# B&R Automation Studio project Project
Automation Studio 4.9

## Configuration Config1

CPU X20CP3586, AutomationRuntime J4.93, Build 4.1.2, Safety 0.0, Vc V4.73.2

### Hardware
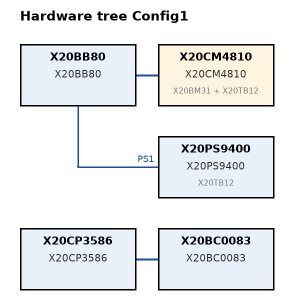
```
X20BB80 : X20BB80 v1.1.0.0
X20BC0083 : X20BC0083 v2.14.0.0  [PLK1 -> X20CP3586.IF3 (NodeNumber=1) [Cable Type=PowerlinkCable, Length=10, Version=1.0.0.3]; SL -> X20BB80.SL1]
  EnableDNA = on
X20BM31 : X20BM31 v1.1.0.0  [X2X1 -> X20BB80.IF1]
X20CM4810 : X20CM4810 v1.7.0.0  [SS1 -> X20TB12a.SS; SL -> X20BM31.SL1]
  Current01 = on
  CalcVel01 = on
  FLOWQ01 = 16#0002
  AICalc01 = on
  AIParameter01 = PEAK
  Current02 = on
X20CP3586 : X20CP3586 v1.10.0.0
  Connector IF2:
    ActivateDevice = 1
    HostName = cotrace-api
    Mode = Manual
    InternetAddress = 10.24.137.37
    SubnetMask = 255.255.255.0
  Connector IF3:
    EplHostName = cotrace-api
    HostName = cotrace-api
  ConfigurationID = CoTrace_Vibor_Config1
  VolatileGlobalPvSize = 200000
  IdleTaskClass = 1
  Cyclic1Duration = 2000
  Cyclic1Tolerance = 2000
  Cyclic3Duration = 48000
  Cyclic3Tolerance = 48000
  Cyclic8Duration = 8000
  Cyclic8Tolerance = 50000000
  Cyclic8Stack = 65000
  FileDevice1
  FileDeviceName1 = BufferData
  FileDevicePath1 = F:/BufferData
  EthernetHostName = cotrace-api
  EthernetDefaultGateway = 10.24.137.1
  FTPProtocol = 3
  FtpUser1
  FtpUsername1 = user
  FtpUserPassword1 = ztK7XSEqskzSOCpiuLWoesyAqwvBD/N0feCBZVSbf+w=
  FtpUserSalt1 = 7xprmDrz
  FTPAccessRight1 = 0
  WebServerProtocol = 2
  ActivateOpcUa = 1
  OpcUaInformationModels_PV_Version = 1
X20PS9400 : X20PS9400 v1.8.0.0  [SS1 -> X20TB12.SS; PS -> X20BB80.PS1]
X20TB12 : X20TB12 v1.0.0.0
X20TB12a : X20TB12 v1.0.0.0
```

### Hardware.hw.as4
```
Module X20BB80 (Type=X20BB80, Version=1.1.0.0)
Module X20BC0083 (Type=X20BC0083, Version=2.15.0.0)
  Connection (Connector=PLK1, TargetModule=X20CP3586, TargetConnector=IF3, NodeNumber=1)
    Cable (Type=PowerlinkCable, Length=10, Version=1.0.0.3)
  Connection (Connector=SL, TargetModule=X20BB80, TargetConnector=SL1)
Module X20BM31 (Type=X20BM31, Version=1.1.0.0)
  Connection (Connector=X2X1, TargetModule=X20BB80, TargetConnector=IF1)
Module X20CM4810 (Type=X20CM4810, Version=1.7.0.0)
  Connection (Connector=SS1, TargetModule=X20TB12a, TargetConnector=SS)
  Connection (Connector=SL, TargetModule=X20BM31, TargetConnector=SL1)
  Current01 = on
  CalcVel01 = on
  FLOWQ01 = 16#0002
  AICalc01 = on
  AIParameter01 = PEAK
  Current02 = on
Module X20CP3586 (Type=X20CP3586, Version=1.10.0.0)
  Connector IF2:
    ActivateDevice = 1
    HostName = cotrace-api
    Mode = Manual
    InternetAddress = 10.24.137.37
    SubnetMask = 255.255.255.0
  Connector IF3:
    EplHostName = cotrace-api
    HostName = cotrace-api
  ConfigurationID = CoTrace_Vibor_Config1
  Cyclic8Stack = 64000
  FileDevice1
  FileDeviceName1 = CoTraceWebApiFolder
  FileDevicePath1 = F:/CoTraceWebApiFolder
  FileDevice2
  FileDeviceName2 = SvgData
  FileDevicePath2 = F:/SvgData
  EthernetHostName = cotrace-api
  EthernetDefaultGateway = 10.24.137.1
  FTPProtocol = 3
  FtpUser1
  FtpUsername1 = user
  FtpUserPassword1 = ztK7XSEqskzSOCpiuLWoesyAqwvBD/N0feCBZVSbf+w=
  FtpUserSalt1 = 7xprmDrz
  FTPAccessRight1 = 0
  WebServerProtocol = 2
  ActivateOpcUa = 1
  OpcUaInformationModels_PV_Version = 1
Module X20PS9400 (Type=X20PS9400, Version=1.8.0.0)
  Connection (Connector=SS1, TargetModule=X20TB12, TargetConnector=SS)
  Connection (Connector=PS, TargetModule=X20BB80, TargetConnector=PS1)
Module X20TB12 (Type=X20TB12, Version=1.0.0.0)
Module X20TB12a (Type=X20TB12, Version=1.0.0.0)
```

### IoMap.iom - X20CP3586/IoMap.iom
```iecst
VAR_CONFIG
	::GetBuffer:fubCM4810.ioMapping.BufferInputSequence01 AT %IB."X20CM4810".BufferInputSequence01;
	::GetBuffer:fubCM4810.ioMapping.BufferRxByte01 AT %IB."X20CM4810".BufferRxByte01;
	::GetBuffer:fubCM4810.ioMapping.BufferRxByte02 AT %IB."X20CM4810".BufferRxByte02;
	::GetBuffer:fubCM4810.ioMapping.BufferRxByte03 AT %IB."X20CM4810".BufferRxByte03;
	::GetBuffer:fubCM4810.ioMapping.BufferRxByte04 AT %IB."X20CM4810".BufferRxByte04;
	::GetBuffer:fubCM4810.ioMapping.BufferRxByte05 AT %IB."X20CM4810".BufferRxByte05;
	::GetBuffer:fubCM4810.ioMapping.BufferOutputSequence01 AT %QB."X20CM4810".BufferOutputSequence01;
	::GetBuffer:fubCM4810.ioMapping.BufferTxByte01 AT %QB."X20CM4810".BufferTxByte01;
	::GetBuffer:fubCM4810.ioMapping.BufferTxByte02 AT %QB."X20CM4810".BufferTxByte02;
	::GetBuffer:fubCM4810.ioMapping.BufferTxByte03 AT %QB."X20CM4810".BufferTxByte03;
	::GetBuffer:fubCM4810.ioMapping.BufferTxByte04 AT %QB."X20CM4810".BufferTxByte04;
	::GetBuffer:fubCM4810.ioMapping.BufferLockValid01 AT %IX."X20CM4810".BufferLockValid01;
	::GetBuffer:fubCM4810.ioMapping.RequestBufferLock01 AT %QX."X20CM4810".RequestBufferLock01; (* SensorData[1] - CM4810 Channel 1 *)
	::SensorData[1].RmsAccRaw AT %ID."X20CM4810".RmsAccRaw01;
	::SensorData[1].RmsAccEnvelope AT %ID."X20CM4810".RmsAccEnvelope01;
	::SensorData[1].RmsVelRaw AT %ID."X20CM4810".RmsVelRaw01;
	::SensorData[1].RmsVelEnvelope AT %ID."X20CM4810".RmsVelEnvelope01;
	::SensorData[1].KurtosisRaw AT %ID."X20CM4810".KurtosisRaw01;
	::SensorData[1].SkewnessRaw AT %ID."X20CM4810".SkewnessRaw01;
	::SensorData[1].Vdi3832KtRaw AT %ID."X20CM4810".Vdi3832KtRaw01;
	::SensorData[1].ActSpeed AT %ID."X20CM4810".ActSpeed01;
	::SensorData[2].RmsAccRaw AT %ID."X20CM4810".RmsAccRaw02;
	::SensorData[2].RmsAccEnvelope AT %ID."X20CM4810".RmsAccEnvelope02;
	::SensorData[2].RmsVelRaw AT %ID."X20CM4810".RmsVelRaw02;
	::SensorData[2].RmsVelEnvelope AT %ID."X20CM4810".RmsVelEnvelope02;
	::SensorData[2].KurtosisRaw AT %ID."X20CM4810".KurtosisRaw02;
	::SensorData[2].SkewnessRaw AT %ID."X20CM4810".SkewnessRaw02;
	::SensorData[2].Vdi3832KtRaw AT %ID."X20CM4810".Vdi3832KtRaw02;
	::SensorData[2].ActSpeed AT %ID."X20CM4810".ActSpeed02;
	::SensorData[3].RmsAccRaw AT %ID."X20CM4810".RmsAccRaw03; (*RMS Value of the acceleration raw signal from MinFrequencyRaw to MaxFrequencyRaw [mg], channel 2*)
	::SensorData[3].RmsVelEnvelope AT %ID."X20CM4810".RmsVelEnvelope03; (*RMS Value of the velocity envelope signal from MinFrequencyEnvelope to MaxFrequencyEnvelope [mm/s], channel 3 (0 = calculation of velocity signal is disabled)*)
	::SensorData[3].KurtosisRaw AT %ID."X20CM4810".KurtosisRaw03; (*Kurtosis (4th statistical moment) of the raw signal from 0 Hz to MaxFrequencyRaw [1], channel 3*)
	::SensorData[3].Vdi3832KtRaw AT %ID."X20CM4810".Vdi3832KtRaw03; (*Ratio of the refernce values to the actual measured values of the raw signal as defined in VDI 3832 [1], channel 3*)
	::SensorData[3].SkewnessRaw AT %ID."X20CM4810".SkewnessRaw03; (*Skewnes (3rd statistical moment) of the raw signal from 0 Hz to MaxFrequencyRaw [1], channel 3*)
	::SensorData[3].RmsAccEnvelope AT %ID."X20CM4810".RmsAccEnvelope03; (*RMS Value of the acceleration envelope signal from MinFrequencyEnvelope to MaxFrequencyEnvelope [mg], channel 2*)
	::SensorData[3].RmsVelRaw AT %ID."X20CM4810".RmsVelRaw03; (*RMS Value of the velocity raw signal from MinFrequencyRaw to MaxFrequencyRaw [mm/s], channel 2 (0 = calculation of velocity signal is disabled)*)
	::SensorData[4].RmsAccRaw AT %ID."X20CM4810".RmsAccRaw04;
	::SensorData[4].RmsAccEnvelope AT %ID."X20CM4810".RmsAccEnvelope04;
	::SensorData[4].RmsVelRaw AT %ID."X20CM4810".RmsVelRaw04;
	::SensorData[4].RmsVelEnvelope AT %ID."X20CM4810".RmsVelEnvelope04;
	::SensorData[4].KurtosisRaw AT %ID."X20CM4810".KurtosisRaw04;
	::SensorData[4].SkewnessRaw AT %ID."X20CM4810".SkewnessRaw04;
	::SensorData[4].Vdi3832KtRaw AT %ID."X20CM4810".Vdi3832KtRaw04;
	::SensorData[1].ActSpeed AT %QD."X20CM4810".ActSpeed01;
	::SensorData[2].ActSpeed AT %QD."X20CM4810".ActSpeed02;
	::SensorData[3].ActSpeed AT %QD."X20CM4810".ActSpeed03;
	::SensorData[4].ActSpeed AT %QD."X20CM4810".ActSpeed04;
END_VAR
```

## Logical view

Binary libraries used (declarations not repeated): FileIO, runtime, sys_lib, AsBrStr, AsIOVib, AsFltGen, brsystem, AsIOAcc

### Global.typ - Global data types
```iecst
(* ============================================================ *)
(* CM4810 SENSOR CHANNEL DATA - Mapped from X20CM4810 process data via IoMap *)

TYPE
	SensorChannelData : 	STRUCT
		RmsAccRaw : REAL;			(* RMS acceleration raw [g] *)
		RmsAccEnvelope : REAL;		(* RMS acceleration envelope [g] *)
		RmsVelRaw : REAL;			(* RMS velocity raw [mm/s] *)
		RmsVelEnvelope : REAL;		(* RMS velocity envelope [mm/s] *)
		KurtosisRaw : REAL;			(* Kurtosis raw [-] *)
		SkewnessRaw : REAL;			(* Skewness raw [-] *)
		Vdi3832KtRaw : REAL;		(* VDI3832 Kt raw [-] *)
		ActSpeed : REAL;			(* Actual speed [rpm] *)
	END_STRUCT;
END_TYPE

(* ============================================================ *)
(* CSV EXPORT STATE MACHINE - Single state variable for GetBuffer <-> SaveData communication*)

TYPE
	CSVExportState :
		(
		CSV_IDLE := 0, (* Waiting for export request *)
		CSV_REQUESTED := 1, (* GetBuffer requested export *)
		CSV_PROCESSING := 2, (* SaveData is exporting *)
		CSV_COMPLETED := 3, (* Export done, CSV ready *)
		CSV_ERROR := 4 (* Export failed *)
		);
END_TYPE

(* ============================================================ *)
(* OPC UA COMMAND INTERFACE [API -> PLC] - Write these variables from FastAPI to configure the job*)

TYPE
	BufferUploadCmd : 	STRUCT
		WorkID : STRING[80] := 'debug_123'; (* Unique job ID: "mach5_sens12_1234567890_raw" *)
		ModulePath : STRING[30] := 'IF3.ST1.IF1.ST2'; (* "IF3.ST1.IF1.ST2" - X2X module path *)
		BufferNumber : USINT := 66; (* Buffer to download: 9,11,13,15,25,27,29,31,66,67,70,71... *)
		BufferLength : UDINT := 4097; (* Number of values: 4097, 8193, or 65535 *)
		Start : BOOL := 0; (* Edge trigger - set TRUE to start job *)
		Reset : BOOL := 0; (* Edge trigger - set TRUE to reset after Done *)
	END_STRUCT;
END_TYPE

(* ============================================================ *)
(* OPC UA STATUS INTERFACE [PLC -> API] - Read these variables from FastAPI to monitor job progress*)

TYPE
	BufferUploadStatus : 	STRUCT
		CurrentWorkID : STRING[80]; (* Currently processing WorkID *)
		Busy : BOOL := 0; (* TRUE when PLC is working on a job *)
		Done : BOOL := 0; (* TRUE when job completed (CSV ready on FTP) *)
		Error : BOOL := 0; (* TRUE if error occurred *)
		ErrorID : UINT := 0; (* Error code from vbioCM4810.status or custom error *)
		Progress : USINT := 0; (* Job progress: 0-100% *)
		CSVFileName : STRING[100]; (* Name of generated CSV file *)
	END_STRUCT;
END_TYPE

(* ============================================================ *)
(* MAIN STRUCTURE - Global variable gTrace*)

TYPE
	TraceVibro : 	STRUCT  (* OPC UA Interface - API <-> PLC *)
		BufferUpload : BufferUploadCmd;
		BufferStatus : BufferUploadStatus; (* Internal communication - GetBuffer <-> SaveData *)
		CSVExport : CSVExportState; (* Single state variable: IDLE/REQUESTED/PROCESSING/COMPLETED/ERROR *) (* Buffer data storage - max 8193 values *) (* Note: Most CM4810 buffers use 8193 values. Only special cases use 65535. *)
		xAxis : ARRAY[0..8192]OF REAL;
		yAxis : ARRAY[0..8192]OF REAL;
	END_STRUCT;
END_TYPE
```

### Global.var - Global variables
```iecst
VAR
	gTrace : TraceVibro;
	SensorData : ARRAY[1..4] OF SensorChannelData;
END_VAR
```


### Program Logical/VibroBuffer/GetBuffer (IEC)

#### Variables.var
```iecst
VAR
	fubCM4810 : vbioCM4810; (* Function block for accessing the buffers of a CM4810 module *)
	bInitialized : BOOL := FALSE;
	stMachine : UINT := 0; (* Status of the main state machine *)
	i : INT;
END_VAR
```

#### Main.st
```iecst
PROGRAM _INIT
	(* Enable function block *)
	fubCM4810.enable := TRUE;

	(* Set array pointers - these stay constant *)
	fubCM4810.paramBufferUpload.pArrayXaxis := ADR(gTrace.xAxis);
	fubCM4810.paramBufferUpload.pArrayYaxis := ADR(gTrace.yAxis);

	(* Module path pointer - points directly to OPC UA BufferUpload structure *)
	fubCM4810.paramMain.pModulePath := ADR(gTrace.BufferUpload.ModulePath);

	(* Initialize SensorData - clear all channels [1..4] *)
	FOR i := 1 TO 4 DO
		SensorData[i].RmsAccRaw := 0.0;
		SensorData[i].RmsAccEnvelope := 0.0;
		SensorData[i].RmsVelRaw := 0.0;
		SensorData[i].RmsVelEnvelope := 0.0;
		SensorData[i].KurtosisRaw := 0.0;
		SensorData[i].SkewnessRaw := 0.0;
		SensorData[i].Vdi3832KtRaw := 0.0;
		SensorData[i].ActSpeed := 0.0;
	END_FOR;

	(* NOTE: BufferNumber, BufferLength configured dynamically in _CYCLIC from BufferUpload command *)

END_PROGRAM

PROGRAM _CYCLIC
	(* First scan initialization - runs once after download *)
	IF NOT bInitialized THEN
		stMachine := 0;
		gTrace.BufferStatus.Done := FALSE;
		gTrace.BufferStatus.Busy := FALSE;
		gTrace.BufferStatus.Error := FALSE;
		gTrace.BufferStatus.Progress := 0;
		gTrace.BufferStatus.CurrentWorkID := '';
		bInitialized := TRUE;
	END_IF;

	CASE stMachine OF
		0: (* IDLE - Wait for job from API via OPC UA *)
			fubCM4810.requestBufferLock := FALSE;
			fubCM4810.uploadBuffer := FALSE;

			IF gTrace.BufferUpload.Start THEN
				(* Load job configuration from OPC UA *)
				gTrace.BufferStatus.CurrentWorkID := gTrace.BufferUpload.WorkID;

				(* Configure buffer download parameters *)
				fubCM4810.paramBufferUpload.moduleBuffer := gTrace.BufferUpload.BufferNumber;
				fubCM4810.paramBufferUpload.nrArrayElements := gTrace.BufferUpload.BufferLength;

				(* Set status *)
				gTrace.BufferStatus.Busy := TRUE;
				gTrace.BufferStatus.Done := FALSE;
				gTrace.BufferStatus.Error := FALSE;
				gTrace.BufferStatus.Progress := 0;

				(* Reset start trigger *)
				gTrace.BufferUpload.Start := FALSE;

				stMachine := 1;
			END_IF;

		1: (* LOCK BUFFERS *)
			fubCM4810.requestBufferLock := TRUE;
			gTrace.BufferStatus.Progress := 10;

			IF fubCM4810.bufferLockValid = TRUE THEN
				stMachine := 2;
			END_IF;

		2: (* DOWNLOAD BUFFER *)
			fubCM4810.uploadBuffer := TRUE;
			gTrace.BufferStatus.Progress := 50;

			IF fubCM4810.bufferUploadDone = TRUE THEN
				fubCM4810.uploadBuffer := FALSE;
				stMachine := 3;
			END_IF;

		3: (* TRIGGER CSV EXPORT *)
			gTrace.CSVExport := CSV_REQUESTED;
			gTrace.BufferStatus.Progress := 70;
			stMachine := 4;

		4: (* WAIT FOR CSV COMPLETION *)
			IF gTrace.CSVExport = CSV_COMPLETED THEN
				gTrace.CSVExport := CSV_IDLE;  (* Reset for next job *)
				stMachine := 5;
			ELSIF gTrace.CSVExport = CSV_ERROR THEN
				(* CSV export failed *)
				gTrace.BufferStatus.Error := TRUE;
				gTrace.BufferStatus.ErrorID := 9000;  (* Custom error: CSV export failed *)
				gTrace.CSVExport := CSV_IDLE;
				stMachine := 5;
			END_IF;

		5: (* UNLOCK BUFFERS *)
			fubCM4810.requestBufferLock := FALSE;
			gTrace.BufferStatus.Progress := 90;

			IF fubCM4810.bufferLockValid = FALSE THEN
				gTrace.BufferStatus.Progress := 100;
				gTrace.BufferStatus.Done := TRUE;
				gTrace.BufferStatus.Busy := FALSE;
				stMachine := 6;
			END_IF;

		6: (* COMPLETED - Wait for Reset from API *)
			IF gTrace.BufferUpload.Reset THEN
				gTrace.BufferStatus.Done := FALSE;
				gTrace.BufferStatus.Busy := FALSE;
				gTrace.BufferStatus.Progress := 0;
				gTrace.BufferStatus.CurrentWorkID := '';
				gTrace.BufferUpload.Reset := FALSE;
				stMachine := 0;
			END_IF;
	END_CASE;

	(* Update error status *)
	IF fubCM4810.status <> 0 THEN
		gTrace.BufferStatus.Error := TRUE;
		gTrace.BufferStatus.ErrorID := fubCM4810.status;
	ELSE
		gTrace.BufferStatus.Error := FALSE;
		gTrace.BufferStatus.ErrorID := 0;
	END_IF;

	(* Execute function block *)
	fubCM4810();

END_PROGRAM

PROGRAM _EXIT
	(* Insert code here *)

END_PROGRAM
```

### Program Logical/VibroBuffer/SaveData (IEC)

#### Variables.var
```iecst
(* CSV Export Variables *)
VAR CONSTANT
	CRLF : STRING[4] := '$r$n'; (* Carriage Return + Line Feed *)
	FILE_DEVICE : STRING[20] := 'BufferData'; (* FTP file device *)
	BUFFER_SIZE_LIMIT : UDINT := 60000; (* Write to file when buffer reaches 60KB *)
	BATCH_SIZE : UINT := 500; (* Number of rows to process per cycle *)
END_VAR
(* State machine *)
VAR
	fileStep : UINT := 0; (* File operations *)
	fileName : STRING[255]; (* Dynamic CSV filename from WorkID *)
	fbFileCreate : FileCreate;
	fbFileWrite : FileWrite;
	fbFileClose : FileClose;
	FDelete : FileDelete; (* Buffer for batch CSV writing *)
	fileBuffer : STRING[65535];
	rowIndex : UINT;
	StartAddress : UDINT;
	NextAddress : UDINT;
	batchCounter : UINT;
END_VAR
```

#### Main.st
```iecst
PROGRAM _INIT
	(* No initialization needed - all configuration comes from gTrace.BufferUpload *)
END_PROGRAM

PROGRAM _CYCLIC
	(* CSV File Writing State Machine *)
	CASE fileStep OF
		0: (* Wait for trigger *)
			IF gTrace.CSVExport = CSV_REQUESTED THEN
				gTrace.CSVExport := CSV_PROCESSING;

				(* Generate dynamic filename from WorkID *)
				fileName := gTrace.BufferStatus.CurrentWorkID;
				brsstrcat(ADR(fileName), ADR('.csv'));

				fileStep := 10;
			END_IF;

		10: (* Delete existing file if it exists *)

			FDelete.enable  := TRUE;
			FDelete.pDevice := ADR(FILE_DEVICE);
			FDelete.pName   := ADR(fileName);
			FDelete();

			(* Status: 0=deleted successfully, 20708=file doesn't exist (both OK) *)
			IF (FDelete.status = 0) OR (FDelete.status = 20708) THEN
				fileStep := 20;
			ELSIF (FDelete.status <> 65535) THEN
				(* Real error occurred *)
				gTrace.CSVExport := CSV_ERROR;
				fileStep := 60;
			END_IF

		20: (* Create file *)
			fbFileCreate.enable := TRUE;
			fbFileCreate.pDevice := ADR(FILE_DEVICE);
			fbFileCreate.pFile := ADR(fileName);
			fbFileCreate();
			IF fbFileCreate.status = 0 THEN
				fbFileWrite.enable := TRUE;
				fbFileWrite.ident := fbFileCreate.ident;
				fbFileWrite.offset := 0;
				fbFileClose.enable := TRUE;
				fbFileClose.ident := fbFileCreate.ident;
				fileStep := 30;
			ELSIF fbFileCreate.status <> 65535 THEN
				(* Error creating file *)
				gTrace.CSVExport := CSV_ERROR;
				fileStep := 60;
			END_IF;

		30: (* Write CSV header and initialize pointer tracking *)
			(* Clear buffer *)
			brsmemset(ADR(fileBuffer), 0, SIZEOF(fileBuffer));

			(* Initialize pointer tracking *)
			StartAddress := ADR(fileBuffer);
			NextAddress := StartAddress;

			(* Write CSV header using pointer tracking *)
			NextAddress := brsstrcpy(NextAddress, ADR('index,xAxis,yAxis'));
			NextAddress := brsmemcpy(NextAddress, ADR(CRLF), SIZEOF(CRLF) - 1);

			(* Write header to file *)
			fbFileWrite.pSrc := StartAddress;
			fbFileWrite.len := NextAddress - StartAddress;
			fbFileWrite();
			IF fbFileWrite.status = 0 THEN
				fbFileWrite.offset := fbFileWrite.offset + fbFileWrite.len;

				(* Reset for data rows *)
				brsmemset(ADR(fileBuffer), 0, SIZEOF(fileBuffer));
				NextAddress := StartAddress;
				rowIndex := 0;
				fileStep := 40;
			ELSIF fbFileWrite.status <> 65535 THEN
				(* Error writing header *)
				gTrace.CSVExport := CSV_ERROR;
				fileStep := 50;
			END_IF;

		40: (* Fill buffer in batches - process multiple rows per cycle *)
			(* Process up to BATCH_SIZE rows per cycle *)
			FOR batchCounter := 0 TO (BATCH_SIZE - 1) DO
				(* Check if we have more rows to process *)
				IF rowIndex < gTrace.BufferUpload.BufferLength THEN
					(* Check buffer size before adding row - safety margin 200 bytes *)
					IF ((NextAddress - StartAddress) < (BUFFER_SIZE_LIMIT - 200)) THEN
						(* Add index *)
						NextAddress := NextAddress + brsitoa(rowIndex, NextAddress);

						(* Add delimiter *)
						NextAddress := brsmemcpy(NextAddress, ADR(','), SIZEOF(',') - 1);

						(* Add xAxis value *)
						NextAddress := NextAddress + brsftoa(gTrace.xAxis[rowIndex], NextAddress);

						(* Add delimiter *)
						NextAddress := brsmemcpy(NextAddress, ADR(','), SIZEOF(',') - 1);

						(* Add yAxis value *)
						NextAddress := NextAddress + brsftoa(gTrace.yAxis[rowIndex], NextAddress);

						(* Add line feed (CRLF) at END of row *)
						NextAddress := brsmemcpy(NextAddress, ADR(CRLF), SIZEOF(CRLF) - 1);

						(* Move to next row *)
						rowIndex := rowIndex + 1;
					ELSE
						(* Buffer is nearly full - exit loop and write to file *)
						EXIT;
					END_IF;
				ELSE
					(* All rows processed - exit loop *)
					EXIT;
				END_IF;
			END_FOR;

			(* After batch processing, check if we need to write buffer or continue *)
			IF ((NextAddress - StartAddress) >= (BUFFER_SIZE_LIMIT - 200)) OR (rowIndex >= gTrace.BufferUpload.BufferLength) THEN
				(* Buffer is full or all rows processed - write to file *)
				fileStep := 45;
			END_IF;

		45: (* Write buffer to file *)
			fbFileWrite.pSrc := StartAddress;
			fbFileWrite.len := NextAddress - StartAddress;
			fbFileWrite();
			IF fbFileWrite.status = 0 THEN
				fbFileWrite.offset := fbFileWrite.offset + fbFileWrite.len;
				fileStep := 46;
			ELSIF fbFileWrite.status <> 65535 THEN
				(* Error writing data *)
				gTrace.CSVExport := CSV_ERROR;
				fileStep := 50;
			END_IF;

		46: (* Check if more rows remain or finish *)
			IF rowIndex < gTrace.BufferUpload.BufferLength THEN
				(* More rows to process - reset buffer and continue *)
				brsmemset(ADR(fileBuffer), 0, SIZEOF(fileBuffer));
				NextAddress := StartAddress;
				fileStep := 40;
			ELSE
				(* All rows written - close file *)
				fileStep := 50;
			END_IF;

		50: (* Close file *)
			fbFileClose();
			IF fbFileClose.status = 0 THEN
				gTrace.CSVExport := CSV_COMPLETED;

				(* Update OPC UA status with CSV filename *)
				gTrace.BufferStatus.CSVFileName := fileName;

				fileStep := 60;
			ELSIF fbFileClose.status <> 65535 THEN
				(* Error closing file *)
				gTrace.CSVExport := CSV_ERROR;
				fileStep := 60;
			END_IF;

		60: (* Reset and return to idle *)
			fbFileCreate.enable := FALSE;
			fbFileWrite.enable := FALSE;
			fbFileClose.enable := FALSE;
			FDelete.enable := FALSE;
			fileStep := 0;
	END_CASE;

END_PROGRAM

PROGRAM _EXIT
	(* Insert code here *)

END_PROGRAM
```
